(* PLC project PLC1, Unknown Unnamed 1 *)
(* stored: creationDateTime 2021-02-24T14:42:08, modificationDateTime 2024-08-08T15:35:29 *)

PROGRAM PLC3
  VAR_INPUT
    level : DINT;
  END_VAR
  VAR_OUTPUT
    pump : BOOL;
  END_VAR
  VAR
    low : BOOL;
    high : BOOL;
    low_3 : DINT := 0;
    high_3 : DINT := 10;
  END_VAR

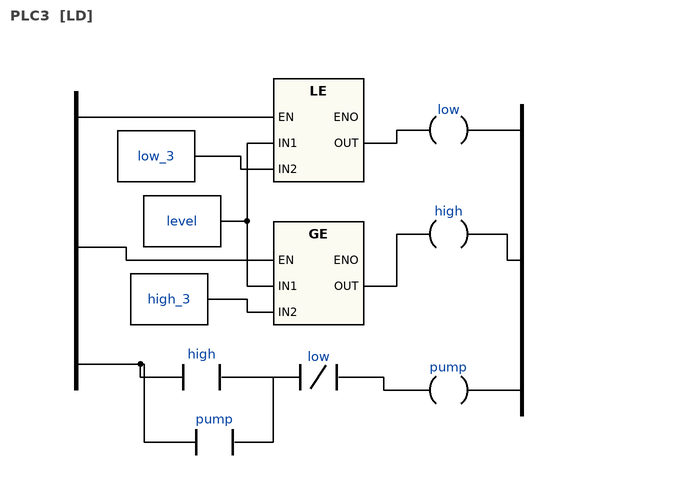
(* LD diagram, written out as Structured Text *)
high := level >= high_3;
low := level <= low_3;
pump := (high OR pump) AND NOT low;
END_PROGRAM

PROGRAM PLC2
  VAR_INPUT
    level : DINT;
  END_VAR
  VAR_OUTPUT
    request : BOOL;
  END_VAR
  VAR
    open_req : BOOL;
    close_req : BOOL;
    low_2 : DINT := 10;
    high_2 : DINT := 20;
  END_VAR

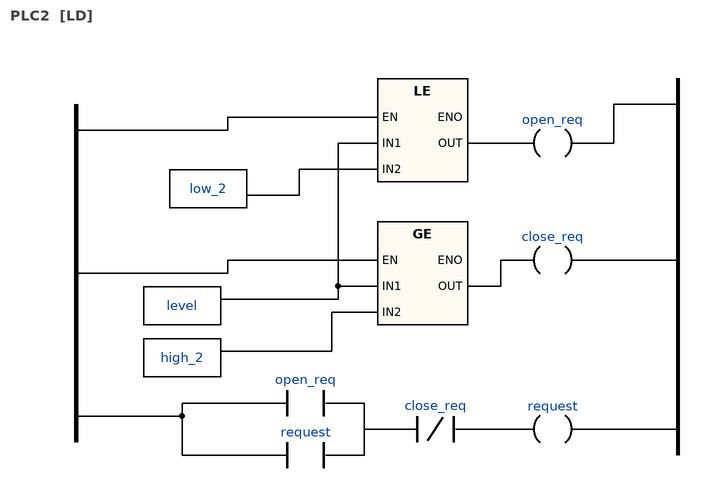
(* LD diagram, written out as Structured Text *)
close_req := level >= high_2;
open_req := level <= low_2;
request := (open_req OR request) AND NOT close_req;
END_PROGRAM

FUNCTION_BLOCK handler_pumps
  VAR_INPUT
    IN1 : DINT;
    IN2 : DINT;
    IN3 : DINT;
  END_VAR
  VAR_OUTPUT
    OUT1 : BOOL;
    OUT2 : BOOL;
  END_VAR
  VAR
    i : INT;
    mytimer : TON;
  END_VAR

            OUT1:=FALSE;
OUT2:=FALSE;
IF IN2 = IN1 then
  OUT1:=TRUE;
END_IF;
IF IN2 = IN3 then
  OUT2:=TRUE;
END_IF;
mytimer(IN := TRUE, PT := t#8000ms);
i:=0;
IF mytimer.Q = TRUE then
   WHILE i<4 do
    OUT1:=TRUE;
  End_WHILE;
End_IF;
 
          
END_FUNCTION_BLOCK

PROGRAM PLC1
  VAR_INPUT
    level : DINT;
    request : DINT;
  END_VAR
  VAR_OUTPUT
    pumps : BOOL;
    valve : BOOL;
  END_VAR
  VAR
    low : BOOL;
    high : BOOL;
    open_req : BOOL;
    close_req : BOOL;
    low_1 : DINT := 40;
    high_1 : DINT := 80;
    handler_pumps0 : handler_pumps;
  END_VAR

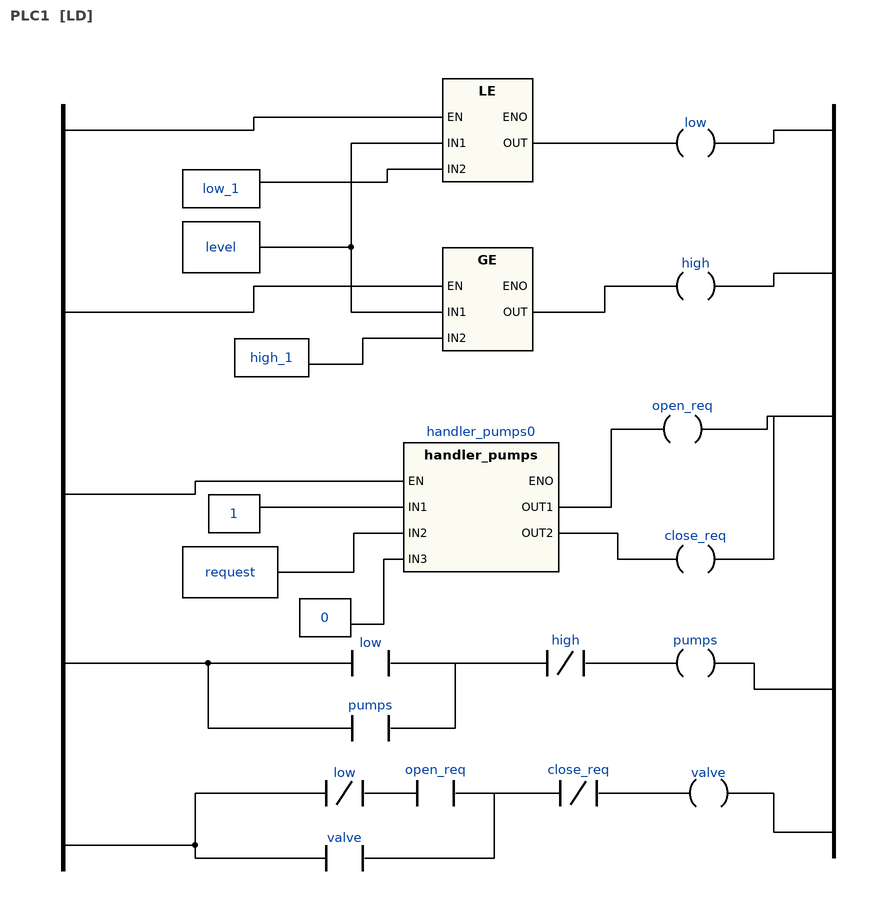
(* LD diagram, written out as Structured Text *)
low := level <= low_1;
high := level >= high_1;
pumps := (low OR pumps) AND NOT high;
valve := (NOT low AND open_req OR valve) AND NOT close_req;
handler_pumps0(IN1 := 1, IN2 := request, IN3 := 0);
open_req := handler_pumps0.OUT1;
close_req := handler_pumps0.OUT2;
END_PROGRAM

CONFIGURATION Config0
  RESOURCE Res0 ON PLC
    TASK task0(INTERVAL := T#20ms, PRIORITY := 0);
    TASK task1(INTERVAL := T#20ms, PRIORITY := 0);
    TASK task2(INTERVAL := T#20ms, PRIORITY := 0);
    PROGRAM instance0 WITH task0 : PLC1;
    PROGRAM instance1 WITH task1 : PLC2;
    PROGRAM instance2 WITH task2 : PLC3;
  END_RESOURCE
END_CONFIGURATION
